{attribute 'GeneratedUsingTerminal: EL7037-0000-0016'}
{attribute addProperty BoxType "EL7037-0000-0016"}
{attribute addProperty Id "EnableBOOL1ResetBOOL1Reduce_torqueBOOL1Digital_output_1BOOL1"}
{attribute addProperty CRC "1607755581"}
{attribute addProperty Size "4"}
TYPE Control_5FD4673D :
STRUCT
	{attribute addProperty Name "Enable"}
	Enable : BOOL;
	{attribute addProperty Name "Reset"}
	Reset : BOOL;
	{attribute addProperty Name "Reduce_torque"}
	Reduce_torque : BOOL;
	{attribute addProperty Name "Digital_output_1"}
	Digital_output_1 : BOOL;
END_STRUCT
END_TYPE

(* stored: Version 1.2.0.0, ProductVersion 3.1.4024.9
   DUT Control_5FD4673D: Id {804b3f6b-9faa-475b-8e35-7e8ca7fa1f11} *)
